(* CODESYS project Cat3.project

Project tree, tasks and I/O mapping:
  Device : CODESYS Control Win V3, 3S - Smart Software Solutions GmbH, order no. 305021, version 3.5.11.0
    application Application
      libraries: Standard, * (System)
      task MainTask (cyclic, interval t#20ms, priority 1) calls PLC_PRG
      task VISU_TASK (cyclic, interval 100 ms, priority 31) calls VisuElems.Visu_Prg
      program PLC_PRG [ST]
      global variables GVL
      function block Plant [ST]
      function block Controller [ST]
      visualisation Visualization
  GlobalImagePool
  text list GlobalTextList
*)

// Device/Application/GVL
{attribute 'qualified_only'}
VAR_GLOBAL
	// Plant only!!!
	IsCatHere : BOOL;
	CatBtn : BOOL;
	CatWeight : REAL := 3.5;
	// --------
	AirQuality : REAL;
	
	SetTimerBtn : BOOL;
	NewTimeInput : INT := 0;

	ClearWeight : REAL := 0.0;
	Weight : REAL := 0.0;	

	CalibrationBtn : BOOL;
	CleanBtn : BOOL;
	
	// --- separator ---
	SepMotor : BOOL;
	SepPosition : REAL := 0.0;
	SepUpped : BOOL := FALSE;
	SepDowned : BOOL := TRUE;
	
	// --- door ---
	DoorLockActuator : BOOL;
	DoorPosition : REAL := 0.0;
	DoorOpened : BOOL := TRUE;
	DoorClosed : BOOL := FALSE;
	
	// --- wastes bin ---
	WastesLevel : REAL := 0.0;
	EmptyWastesBtn : BOOL;
	
	// --- UV ---
	UVLamp : BOOL := FALSE;
	
	// --- aroma ---
	Aroma : BOOL := FALSE;
	AromaLevel : REAL := 100.0;
	RefillAromaBtn : BOOL;
	
	// === LEDS ===
	LowFillerLed : BOOL := FALSE;
	CalibrationModeLed : BOOL := FALSE;
	AromaLed : BOOL := FALSE;
	FullWastesLed : BOOL := FALSE;
	LowAromaLed : BOOL := FALSE;
	
END_VAR

// Device/Application/PLC_PRG
PROGRAM PLC_PRG
VAR
	PlantTask : Plant();
	ControllerTask : Controller();
END_VAR

PlantTask();
ControllerTask();

END_PROGRAM

// Device/Application/Plant
FUNCTION_BLOCK Plant
VAR_INPUT
END_VAR
VAR_OUTPUT
END_VAR
VAR	
	// --- weight ---
	Weight : REAL;
	ClearWeight : REAL;
	WastesLevel : REAL;
	EmptyWastesRE : R_TRIG;
	// ---
	CatWeight : REAL;
	FillerCoast : REAL := 0.05;
	AddedWastes : REAL := 20.0;
	
	// --- aroma ---
	Aroma : BOOL;
	AromaLevel : REAL;
	AromaPart : REAL := 30.0;
	AromaFE : F_TRIG;
	AromaRefillRE : R_TRIG;
	
	// --- cat ---
	CatRE : R_TRIG;

	// --- door ---
	DoorLockActuator : BOOL;
	DoorPosition : REAL;
	DoorLockActuatorRE : R_TRIG;
	DoorLockActuatorFE : F_TRIG;
	// status
	DoorOpening : BOOL := FALSE;
	DoorClosing : BOOL := FALSE;
	DoorOpened : BOOL := TRUE;
	DoorClosed : BOOL := FALSE;
	// controls
	DoorClosedValue : REAL := 250.0;
	DoorOpenedValue : REAL := 0.0;
	DoorMoveStep : REAL := 2.0;
	
	// --- separator ---
	SepMotor : BOOL;
	SepPosition : REAL;
	SepMotorRE : R_TRIG;
	SepMotorFE : F_TRIG;
	// status
	SepUpping : BOOL := FALSE;
	SepDowning : BOOL := FALSE;
	SepUpped : BOOL := FALSE;
	SepUppedRE : R_TRIG;
	SepDowned : BOOL := TRUE;
	// controls
	SepUp : REAL := -90.0;
	SepDown : REAL := 0.0;
	SepMoveStep : REAL := 1.0;
	
END_VAR

// === START ===
// --- weight ---
Weight := GVL.Weight;
ClearWeight := GVL.ClearWeight;
CatWeight := GVL.CatWeight;
WastesLevel := GVL.WastesLevel;
// --- door ---
DoorLockActuator := GVL.DoorLockActuator;
DoorPosition := GVL.DoorPosition;
// --- separator ---
SepMotor := GVL.SepMotor;
SepPosition := GVL.SepPosition;
// --- aroma ---
Aroma := GVL.Aroma;
AromaLevel := GVL.AromaLevel;

// === TRIGGERS ===
CatRE(CLK := GVL.CatBtn);
DoorLockActuatorRE(CLK := DoorLockActuator);
DoorLockActuatorFE(CLK := DoorLockActuator);
SepMotorRE(CLK := SepMotor);
SepMotorFE(CLK := SepMotor);

SepUppedRE(CLK := SepUpped);
AromaFE(CLK := Aroma);

EmptyWastesRE(CLK := GVL.EmptyWastesBtn);
AromaRefillRE(CLK := GVL.RefillAromaBtn);


// === MAIN ===
Weight := ClearWeight;

IF EmptyWastesRE.Q THEN
	WastesLevel := 0.0;
END_IF

IF AromaRefillRE.Q THEN
	AromaLevel := 100.0;
END_IF

// --- cat control ---
IF CatRE.Q AND NOT (DoorClosed OR DoorClosing) THEN
	GVL.IsCatHere := NOT GVL.IsCatHere;
END_IF

IF GVL.IsCatHere THEN
	Weight := ClearWeight + CatWeight;
END_IF

// --- door control ---
IF DoorLockActuatorRE.Q THEN
	DoorClosing := TRUE;
	DoorOpening := FALSE;
ELSIF DoorLockActuatorFE.Q THEN
	DoorOpening := TRUE;
	DoorClosing := FALSE;
END_IF
// Opening
IF DoorPosition - DoorMoveStep >= DoorOpenedValue THEN
	IF DoorOpening AND SepDowned THEN
		DoorPosition := DoorPosition - DoorMoveStep;
	END_IF
	DoorOpened := FALSE;
ELSE
	DoorOpened := TRUE;
	GVL.DoorPosition := DoorOpenedValue;
END_IF
// Closing
IF DoorPosition + DoorMoveStep <= DoorClosedValue THEN
	IF DoorClosing AND SepDowned THEN
		DoorPosition := DoorPosition + DoorMoveStep;
	END_IF
	DoorClosed := FALSE;
ELSE
	DoorClosed := TRUE;
	DoorPosition := DoorClosedValue;
END_IF
IF DoorOpened THEN
	DoorClosed := FALSE;
ELSIF DoorClosed THEN
	DoorOpened := FALSE;
END_IF

// --- separator control ---
IF SepMotorRE.Q THEN
	SepUpping := TRUE;
	SepDowning := FALSE;
ELSIF SepMotorFE.Q THEN
	SepDowning := TRUE;
	SepUpping := FALSE;
END_IF
// Up
IF SepPosition - SepMoveStep >= SepUp THEN
	IF SepUpping AND DoorClosed THEN
		SepPosition := SepPosition - SepMOveStep;
	END_IF
	SepUpped := FALSE;
ELSE
	SepUpped := TRUE;
END_IF
// Down
IF SepPosition + SepMoveStep <= SepDown THEN
	IF SepDowning AND DoorClosed THEN
		SepPosition := SepPosition + SepMoveStep;
	END_IF
	SepDowned := FALSE;
ELSE
	SepDowned := TRUE;
END_IF
IF SepUpped THEN
	SepDowned := FALSE;
ELSIF SepDowned THEN
	SepUpped := FALSE;
END_IF

// --- filler deletion ---
IF SepUppedRE.Q THEN
	IF ClearWeight >= FillerCoast THEN
		ClearWeight := ClearWeight - FillerCoast;
	ELSE
		ClearWeight := 0.0;
	END_IF
	WastesLevel := WastesLevel + AddedWastes;
	IF WastesLevel > 100.0 THEN
		WastesLevel := 100.0;
	END_IF
END_IF

// --- aroma ---
IF AromaFE.Q THEN
	IF AromaLevel >= AromaPart THEN
		AromaLevel := AromaLevel - AromaPart;
	ELSE
		AromaLevel := 0.0;
	END_IF
END_IF


// ============


// === FINAL ===
// --- weight ---
GVL.Weight := Weight;
GVL.ClearWeight := ClearWeight;
GVL.WastesLevel := WastesLevel;
GVL.AromaLevel := AromaLevel;
// --- door ---
GVL.DoorPosition := DoorPosition;
GVL.DoorOpened := DoorOpened;
GVL.DoorClosed := DoorClosed;
// --- separator ---
GVL.SepPosition := SepPosition;
GVL.SepUpped := SepUpped;
GVL.SepDowned := SepDowned;

END_FUNCTION_BLOCK

// Device/Application/Controller
FUNCTION_BLOCK Controller
VAR_INPUT
END_VAR
VAR_OUTPUT
END_VAR
VAR
	FillerWeight : REAL := 0.0;
	LowFillerValue : REAL := 0.5;
	WeightTolerance : REAL := 0.05;
	
	AirQuality : REAL;
	AirQualityThreshold : REAL := 70.0;
	
	VisitsCount : INT := 0;
	VisitsToClean : INT := 1;
	
	NewTime : TIME;

	CalibrationBtnRE : R_TRIG;
	
	// --- aroma ---
	AromaLevel : REAL;
	AromaLowLevel : REAL := 3.0;
	// --- wastes ---
	WastesLevel : REAL;
	WastesCriticalLevel : REAL := 98.0;
	
	// === TIMERS ===
	// --- separating loop ---
	CleaningTimer : TON;
	CleaningDelay : TIME := T#6S;
	// --- cat present ---
	CatWeiter : BOOL := FALSE;
	CatPresentTimer : TON;
	CatPresentDelay : TIME := T#3S;
	// --- UV ---
	UVCleaning : BOOL := FALSE;
	UVCleaningFE : F_TRIG;
	UVTimer : TON;
	UVDelay : TIME := T#5S;
	// --- aroma ---
	Aroma : BOOL := FALSE;
	AromaTimer : TON;
	AromaDelay : TIME := T#2S;
	
	SetTimerBtnRE : R_TRIG;
	ClearBtnRE : R_TRIG;
	CleaningCmd : BOOL := FALSE;
	
	// === FLAGS ===
	Cleaning : BOOL := FALSE;
	CleaningFE : F_TRIG;
	AfterCleaning : BOOL := FALSE;
	AfterUVCleaning : BOOL := FALSE;
	// --- door events ---
	DoorLockActuator : BOOL;
	DoorOpened : BOOL := TRUE;
	DoorOpenedRE : R_TRIG;
	DoorClosed : BOOL := FALSE;
	DoorClosedRE : R_TRIG;
	// --- separator events ---
	SepMotor : BOOL;
	SepUpped : BOOL := FALSE;
	SepDowned : BOOL := TRUE;
	SepUppedRE : R_TRIG;
	SepDownedRE : R_TRIG;
	// --- cat present ---
	IsCatPresent : BOOL := FALSE;
	IsCatPresentRE : R_TRIG;
	IsCatPresentFE : F_TRIG;
	// --- UV ---
	UVLed : BOOL := FALSE;
	// --- aroma ---
	IsAromaLow : BOOL := FALSE;
	AromaLed : BOOL := FALSE;
	// --- low filler ---
	IsFillerLow : BOOL := TRUE;
	IsFillerLowRE : R_TRIG;
	IsFillerLowFE : F_TRIG;
	// --- critical wastes ---
	IsWastesFull : BOOL := FALSE;
	// --- calibration ---
	IsCalibrationMode : BOOL := FALSE;
	IsCalibrationModeRE : R_TRIG;
	IsCalibrationModeFE : F_TRIG;
END_VAR

// === START ===
AromaLevel := GVL.AromaLevel;
WastesLevel := GVL.WastesLevel;
AirQuality := GVL.AirQuality;
DoorOpened := GVL.DoorOpened;
DoorClosed := GVL.DoorClosed;
SepUpped := GVL.SepUpped;
SepDowned := GVL.SepDowned;

SetTimerBtnRE(CLK := GVL.SetTimerBtn);
IF SetTimerBtnRE.Q THEN
	IF GVL.NewTimeInput > 0 THEN
		NewTime := INT_TO_TIME(GVL.NewTimeInput * 1000);
		IF NewTime >= T#500MS THEN
			UVDelay := NewTime;
		END_IF
	END_IF
	GVL.NewTimeInput := TIME_TO_INT(UVDelay) / 1000;
END_IF

// === TRIGGERS ===
CalibrationBtnRE(CLK := GVL.CalibrationBtn);
ClearBtnRE(CLK := GVL.CleanBtn);
DoorOpenedRE(CLK := DoorOpened);
DoorClosedRE(CLK := DoorClosed);
SepUppedRE(CLK := SepUpped);
CleaningFE(CLK := Cleaning);
UVCleaningFE(CLK := UVCleaning);

// === TIMERS ===
CleaningTimer(IN := Cleaning, PT := CleaningDelay);
CatPresentTimer(IN := CatWeiter, PT := CatPresentDelay);
UVTimer(IN := UVCleaning, PT := UVDelay);
AromaTimer(IN := Aroma, PT := AromaDelay);


// === FLAGS ===

// --- low filler
IF FillerWeight < LowFillerValue THEN
	IsFillerLow := TRUE;
ELSE
	IsFillerLow := FALSE;
END_IF

// --- low aroma ---
IF AromaLevel <= AromaLowLevel THEN
	IsAromaLow := TRUE;
ELSE
	IsAromaLow := FALSE;
END_IF

// --- critical wastes ---
IF WastesLevel >= WastesCriticalLevel THEN
	IsWastesFull := TRUE;
ELSE
	IsWastesFull := FALSE;
END_IF

IF ClearBtnRE.Q AND NOT IsFillerLow THEN
	CleaningCmd := TRUE;
END_IF


// === FLAGS TRIGGERS ===
// --- cat present ---
IsCatPresentRE(CLK := IsCatPresent);
IsCatPresentFE(CLK := IsCatPresent);
// --- low filler ---
IsFillerLowRE(CLK := IsFillerLow);
IsFillerLowFE(CLK := IsFillerLow);
// --- calibration ---
IsCalibrationModeRE(CLK := IsCalibrationMode);
IsCalibrationModeFE(CLK := IsCalibrationMode);


// === MAIN ===

// --- calibration ---
IF IsCalibrationMode THEN
	FillerWeight := GVL.Weight;
	IF CalibrationBtnRE.Q THEN
		IsCalibrationMode := FALSE;
	END_IF
ELSE
	IF CalibrationBtnRE.Q AND NOT IsCatPresent AND NOT Cleaning AND NOT UVCleaning AND NOT Aroma THEN
		IsCalibrationMode := TRUE;
	END_IF
END_IF

// --- weight sensor ---
IF (GVL.Weight < FillerWeight) THEN
	FillerWeight := GVL.Weight;
END_IF
IF (GVL.Weight - FillerWeight > WeightTolerance) AND NOT IsFillerLow THEN
	IsCatPresent := TRUE;
	CatWeiter := FALSE;
ELSE
	IsCatPresent := FALSE;
END_IF

// --- cat visits ---
IF IsCatPresentFE.Q AND NOT IsWastesFull THEN
	CatWeiter := TRUE;
END_IF

// After delay starting cleaning
IF CatPresentTimer.Q THEN
	VisitsCount := VisitsCount + 1;
	Cleaning := TRUE;
	DoorLockActuator := TRUE;
	SepMotor := TRUE;
	CatWeiter := FALSE;
END_IF
// Down separator
IF SepUpped AND CleaningTimer.Q THEN
	SepMotor := FALSE;
	DoorLockActuator := FALSE;
	Cleaning := FALSE;
END_IF

IF CleaningFE.Q THEN
	AfterCleaning := TRUE;
END_IF

// --- UV ---
IF AirQuality > AirQualityThreshold THEN
	CleaningCmd := TRUE;
END_IF
IF (VisitsCount > VisitsToClean OR CleaningCmd) AND NOT IsCatPresent THEN
	IF AfterCleaning OR (AirQuality > AirQualityThreshold AND NOT IsCatPresent) OR (CleaningCmd AND NOT IsCatPresent) THEN
		DoorLockActuator := TRUE;
		SepMotor := FALSE;
		IF SepDowned AND DoorClosed THEN
			UVCleaning := TRUE;
		END_IF
	END_IF
ELSE
	AfterCleaning := FALSE;
END_IF

IF UVTimer.Q THEN
	UVCleaning := FALSE;
	DoorLockActuator := FALSE;
	VisitsCount := 0;
	AirQuality := 0.0;
	CleaningCmd := FALSE;
END_IF

IF UVCleaning THEN
	UVLed := TRUE;
ELSE
	UVLed := FALSE;
END_IF

// --- aroma ---
IF UVCleaningFE.Q THEN
	Aroma := TRUE;
END_IF
IF Aroma AND IsAromaLow THEN
	Aroma := FALSE;
	DoorLockActuator := FALSE;
END_IF
IF Aroma THEN
	AromaLed := TRUE;
	DoorLockActuator := TRUE;
	IF AromaTimer.Q THEN
		Aroma := FALSE;
		AromaLed := FALSE;
		DoorLockActuator := FALSE;
	END_IF
END_IF


// --- stop events ---

// --- leds ---
// low filler
GVL.LowFillerLed := IsFillerLow;
// calibration mode
GVL.CalibrationModeLed := IsCalibrationMode;


// ============


// === FINAL ===
GVL.AirQuality := AirQuality;
GVL.DoorLockActuator := DoorLockActuator;
GVL.SepMotor := SepMotor;
GVL.UVLamp := UVLed;
GVL.Aroma := Aroma;
GVL.AromaLed := AromaLed;
GVL.LowAromaLed := IsAromaLow;
GVL.FullWastesLed := IsWastesFull;

END_FUNCTION_BLOCK

// Device/Application/Visualization
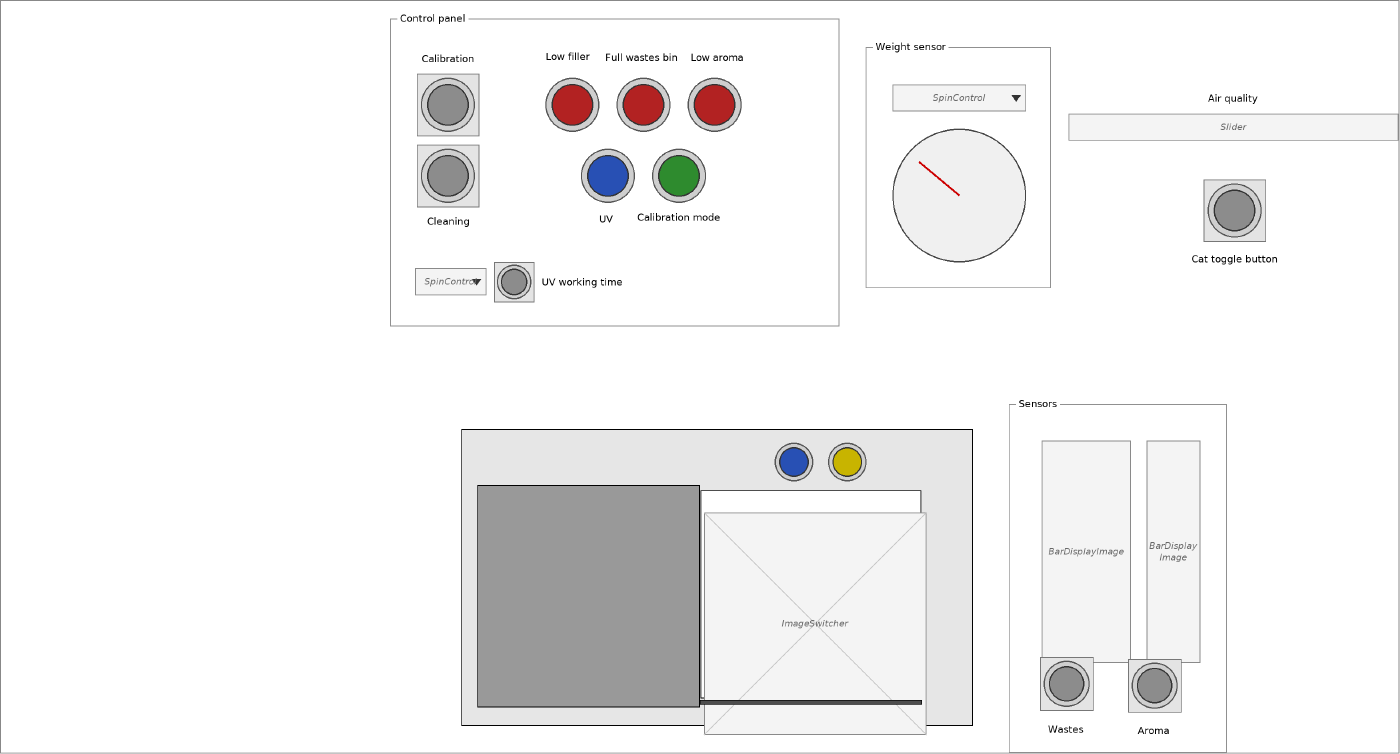
VISUALIZATION Visualization  // 1575x849
    RoundedRectangle (519,483 575x334)
    RoundedRectangle (788,552 248x234)
    ImageSwitcher (792,577 250x250), variable: GVL.IsCatHere, background image: cat, behaviour: TOGGLE
    PushSwitch (1354,202 70x70), variable: GVL.CatBtn, behaviour: TOGGLE, style: Switch-PushSwitch-Gray
    RoundedRectangle (537,546 250x250)
        p3560616238: GVL.DoorPosition
    Rectangle (787,788 250x5)
        p2858320360: GVL.SepPosition
    Lamp1 (868,495 50x50), variable: GVL.UVLamp, style: Lamp-Lamp1-Blue
    Lamp1 (928,495 50x50), variable: GVL.AromaLed, style: Lamp-Lamp1-Yellow
    Slider (1202,128 371x30), variable: GVL.AirQuality, scale 0..100
    GroupBox (439,13 505x354), "Control panel"
        PushSwitch (30,70 70x70), variable: GVL.CalibrationBtn, behaviour: TOGGLE, style: Switch-PushSwitch-Gray
        Lamp1 (170,70 70x70), variable: GVL.LowFillerLed, style: Lamp-Lamp1-Red
        Lamp1 (290,150 70x70), variable: GVL.CalibrationModeLed, style: Lamp-Lamp1-Green
        Lamp1 (210,150 70x70), variable: GVL.UVLamp, style: Lamp-Lamp1-Blue
        Lamp1 (250,70 70x70), variable: GVL.FullWastesLed, style: Lamp-Lamp1-Red
        Lamp1 (330,70 70x70), variable: GVL.LowAromaLed, style: Lamp-Lamp1-Red
        PushSwitch (30,150 70x70), variable: GVL.CleanBtn, behaviour: TOGGLE, style: Switch-PushSwitch-Gray
        Label (123,24 154x54), "Low filler"
        Label (206,25 154x54), "Full wastes bin"
        Label (291,25 154x54), "Low aroma"
        Label (166,207 154x54), "UV"
        Label (248,205 154x54), "Calibration mode"
        Label (6,214 119x45), "Cleaning"
        Label (17,34 96x39), "Calibration"
        SpinControl (28,289 80x30), variable: GVL.NewTimeInput
        PushSwitch (117,282 45x45), variable: GVL.SetTimerBtn, behaviour: TOGGLE, style: Switch-PushSwitch-Gray
        Label (139,278 154x54), "UV working time"
    Label (1312,265 154x54), "Cat toggle button"
    GroupBox (974,45 208x279), "Weight sensor"
        SpinControl (30,50 150x30), variable: GVL.ClearWeight
            p1653691745: 0.2
        Meter360 (30,100 150x150), value: GVL.Weight, style: Meter-Meter360-Gray, scale format: %.1f, scale 0..10
    Label (1310,84 154x54), "Air quality"
    GroupBox (1135,447 245x400), "Sensors"
        BarDisplayImage (155,49 60x250), value: GVL.AromaLevel, style: BarDisplayImage-Gray, scale format: %.1f, scale 0..100
        BarDisplayImage (37,49 100x250), value: GVL.WastesLevel, style: BarDisplayImage-Gray, scale format: %.1f, scale 0..100
        PushSwitch (35,293 60x60), variable: GVL.EmptyWastesBtn, behaviour: TOGGLE, style: Switch-PushSwitch-Gray
        PushSwitch (134,295 60x60), variable: GVL.RefillAromaBtn, behaviour: TOGGLE, style: Switch-PushSwitch-Gray
        Label (124,362 78x28), "Aroma"
        Label (22,361 84x27), "Wastes"
END_VISUALIZATION
